// TIA Portal V18 export
VAR_GLOBAL   // PLC tag table "03 Costanti Nomi Stazioni"
END_VAR
VAR_GLOBAL CONSTANT   // user constants
   "STZ QUADRO" : Int := 1;
   "STZ PROFINET" : Int := 2;
   "STZ GENERALE" : Int := 3;
   "STZ ASPO+CULLA" : Int := 4;
   "STZ RADDRIZZATRICE" : Int := 5;
   "STZ GIUNZIONE" : Int := 6;
   "STZ ALIM" : Int := 7;
   "STZ PLOTTER" : Int := 8;
   "STZ PUNZONATURA" : Int := 9;
   "STZ PROFILA" : Int := 10;
   "STZ TAGLIO" : Int := 11;
   "STZ SCARICO" : Int := 12;
END_VAR
